// TIA Portal V19 export
TYPE "TAx_Fol_Ctrl"
// stored: Access Published
   STRUCT
      SafeStop : Bool;   // 1 = Emergency stop active / Emergency stop (device in safe state)
      Rst : Bool;   // Reset alarms
      RstHW : Bool;   // Reset hardware
      Power : Bool;   // Power axis command
      Homing : Bool;
      VelocityPositionControlled : Bool;
      MovePlus : Bool;
      MoveMinus : Bool;
      MoveAbsolute : Bool;
      GearIn : Bool;
      ExtControl : Bool;   // Axis is controlled from external istruction (MC_Halt not work)
      HomeMode : Int;   // see MC Home
      HomePosition : LReal;
      Velocity : LReal;
      Acceleration : LReal;
      Deceleration : LReal;
      Jerk : LReal;
      MoveAbsTarget : LReal;
      MoveAbsDirection : Int := 3;
      GearInDenominatorRatio : DInt;
      GearInNumeratorRatio : DInt;
   END_STRUCT;
END_TYPE
